FUNCTION_BLOCK hsv2rgb (* Simple helper function, converting HSV color space to RGB color space *)
  (* Standard: 61499-2; Description: Wiki: https://en.wikipedia.org/wiki/HSL_and_HSV *)
  (* Version 1.0, 2022-07-16, franz *)
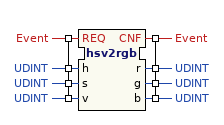
  EVENT_INPUT
    REQ WITH h, s, v; (* Service Request *)
  END_EVENT
  EVENT_OUTPUT
    CNF WITH r, g, b; (* Confirmation of Requested Service *)
  END_EVENT
  VAR_INPUT
    h : UDINT; (* hue *)
    s : UDINT; (* saturation *)
    v : UDINT; (* value *)
  END_VAR
  VAR_OUTPUT
    r : UDINT; (* red *)
    g : UDINT; (* green *)
    b : UDINT; (* blue *)
  END_VAR
END_FUNCTION_BLOCK
